// SIMATIC S7-200 SMART project (STEP 7-Micro/WIN SMART), CPU ST40

SYMBOL_TABLE Table 1
Stop_            V0.0
FACTOR_IO_RUNNING V0.1
Level_meter      VW100
Flow_meter       VW102
Setpoint         VW104
Stop_Light       Q0.0
Fill_Valve       QW2
Discharge_Valve  QW4
SP               QW6
PV               QW8
END_SYMBOL_TABLE

SYMBOL_TABLE System Symbols
Always_On        SM0.0    // Always ON
END_SYMBOL_TABLE

ORGANIZATION_BLOCK MAIN:OB1
TITLE=Program Comments
VAR
PID_Out:WORD;	// LW0 
END_VAR
BEGIN
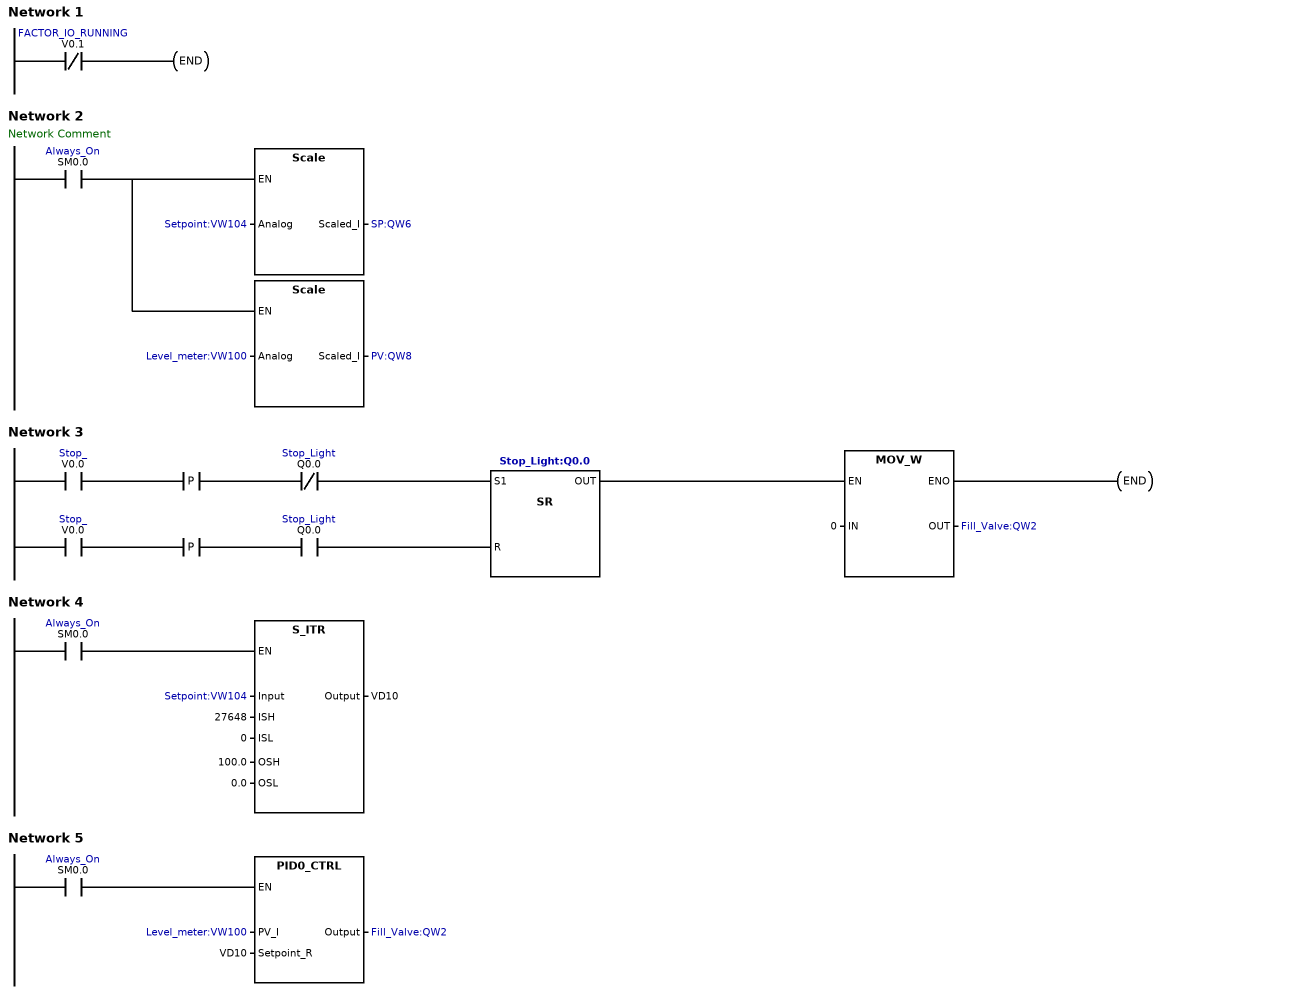
Network 1
LDN    FACTOR_IO_RUNNING:V0.1
END
Network 2
// Network Comment
LD     Always_On:SM0.0
CALL   Scale:SBR0, Setpoint:VW104, SP:QW6
CALL   Scale:SBR0, Level_meter:VW100, PV:QW8
Network 3
LD     Stop_:V0.0
EU
AN     Stop_Light:Q0.0
LD     Stop_:V0.0
EU
A      Stop_Light:Q0.0
NOT
A      Stop_Light:Q0.0
OLD
=      Stop_Light:Q0.0
MOVW   0, Fill_Valve:QW2
AENO
END
Network 4
LD     Always_On:SM0.0
CALL   S_ITR:SBR1, Setpoint:VW104, 27648, 0, 100.0, 0.0, VD10
Network 5
LD     Always_On:SM0.0
CALL   PID0_CTRL:SBR3, Level_meter:VW100, VD10, Fill_Valve:QW2
END_ORGANIZATION_BLOCK

SUBROUTINE_BLOCK Scale:SBR0
TITLE=Subroutine Comments
VAR_INPUT
Analog:WORD;	// LW0 
END_VAR
VAR_OUTPUT
Scaled_I:INT;	// LW2 
END_VAR
VAR
Scaled_R_D_1:REAL;	// LD4 
Scaled_R_D_2:DWORD;	// LD8 
END_VAR
BEGIN
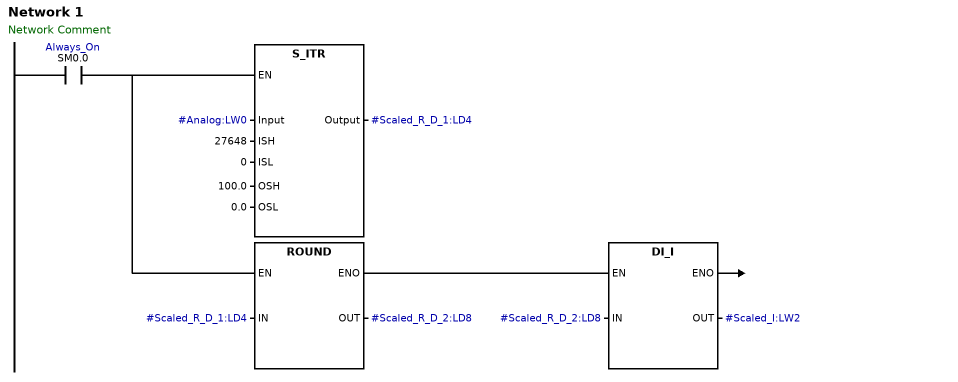
Network 1
// Network Comment
LD     Always_On:SM0.0
CALL   S_ITR:SBR1, #Analog:LW0, 27648, 0, 100.0, 0.0, #Scaled_R_D_1:LD4
ROUND  #Scaled_R_D_1:LD4, #Scaled_R_D_2:LD8
AENO
DTI    #Scaled_R_D_2:LD8, #Scaled_I:LW2
Network 2
// Network Comment
END_SUBROUTINE_BLOCK

// SBR1: protected block, not included

// SBR2: protected block, not included

// SBR3: protected block, not included

// INT1: protected block, not included
